TYPE Channel_830843C1 EXTENDS DigitalInputBase:
STRUCT
	{attribute addProperty Name "Input"}
	Input AT %I* : BOOL;
END_STRUCT
END_TYPE

(* stored: Version 1.1.0.1, ProductVersion 3.1.4024.9
   DUT Channel_830843C1: Id {f9811457-04e6-0b1e-2800-2afd8b1b50a8} *)
